    rq_activate_all_grippers(False)
    # end: URCap Program Node
    $ 3 "Wait: 10.0"
    sleep(10.0)
    # begin: URCap Program Node
    #   Source: Robotiq_Grippers, 1.8.0.1, Robotiq Inc.
    #   Type: Gripper
    $ 4 "Gripper Open (1)"
    if not(gripper_connected[0]):
      popup("Gripper 1 must be connected to run this program.", "No connection", False, True, True)
    end
    if not(rq_is_gripper_activated("1")):
      popup("Gripper 1 is not activated. Go to Installation tab > Gripper to activate it and run the program again.", "Not activated", False, True, True)
    end
    rq_set_pos_spd_for(0, 41, 66, "1")
    rq_wait_pos_spe_for_request(0, 41, 66, "1")
    rq_go_to("1")
    rq_wait("1")
    # end: URCap Program Node
    $ 5 "Loop 20 times"
    Loop_1 = 0
    while (Loop_1 < 20):
      $ 6 "MoveJ"
      $ 7 "start_position"
      movej(get_inverse_kin(p[.170260721946, .070237990876, .680621912575, .161854371436, 1.656832500967, -.237542251413], qnear=[-3.4132304827319544, -1.5469310919391077, 0.21133089065551758, -1.7181108633624476, -1.552213493977682, 7.7919034401523035]), a=1.3962634015954636, v=1.0471975511965976)
      $ 8 "MoveJ"
      $ 9 "backcase_pos"
      movej(get_inverse_kin(p[.279895687381, -.152872741101, .176453276827, .147115205195, -3.063448562531, .021495505714], qnear=[-3.980655018483297, -1.3704388777362269, 2.021009922027588, -2.1860244909869593, -1.6399787108050745, 6.916248623524801]), a=1.3962634015954636, v=1.0471975511965976)
      # begin: URCap Program Node
      #   Source: Robotiq_Grippers, 1.8.0.1, Robotiq Inc.
      #   Type: Gripper
      $ 10 "Gripper Close (1)"
      if not(gripper_connected[0]):
        popup("Gripper 1 must be connected to run this program.", "No connection", False, True, True)
      end
      if not(rq_is_gripper_activated("1")):
        popup("Gripper 1 is not activated. Go to Installation tab > Gripper to activate it and run the program again.", "Not activated", False, True, True)
      end
      rq_set_pos_spd_for(255, 41, 66, "1")
      rq_wait_pos_spe_for_request(255, 41, 66, "1")
      rq_go_to("1")
      rq_wait("1")
      # end: URCap Program Node
      # begin: URCap Program Node
      #   Source: Robotiq_Grippers, 1.8.0.1, Robotiq Inc.
      #   Type: Grip Check
      $ 11 "Grip Check"
      # begin: URCap Program Node
      #   Source: Robotiq_Grippers, 1.8.0.1, Robotiq Inc.
      #   Type: If
      $ 12 "If object detected          "
      if (rq_is_object_detected(1)):
        $ 13 "release_pos"
        movej(get_inverse_kin(p[.470773091472, .179206339821, .406393760794, -.295071821076, 2.303841954291, .069768841993], qnear=[-3.0107629934894007, -0.39652759233583623, -0.4139049688922327, -1.5799277464496058, -1.5207040945636194, 7.751115862523214]), a=1.3962634015954636, v=1.0471975511965976)
        # begin: URCap Program Node
        #   Source: Robotiq_Grippers, 1.8.0.1, Robotiq Inc.
        #   Type: Gripper
        $ 14 "Gripper Open (1)"
        if not(gripper_connected[0]):
          popup("Gripper 1 must be connected to run this program.", "No connection", False, True, True)
        end
        if not(rq_is_gripper_activated("1")):
          popup("Gripper 1 is not activated. Go to Installation tab > Gripper to activate it and run the program again.", "Not activated", False, True, True)
        end
        rq_set_pos_spd_for(0, 66, 41, "1")
        rq_wait_pos_spe_for_request(0, 66, 41, "1")
        rq_go_to("1")
        rq_wait("1")
        # end: URCap Program Node
        # end: URCap Program Node
        # begin: URCap Program Node
        #   Source: Robotiq_Grippers, 1.8.0.1, Robotiq Inc.
        #   Type: Else
        $ 15 "Else"
      else:
        # begin: URCap Program Node
        #   Source: Robotiq_Grippers, 1.8.0.1, Robotiq Inc.
        #   Type: Gripper
        $ 16 "Gripper Open (1)"
        if not(gripper_connected[0]):
          popup("Gripper 1 must be connected to run this program.", "No connection", False, True, True)
        end
        if not(rq_is_gripper_activated("1")):
          popup("Gripper 1 is not activated. Go to Installation tab > Gripper to activate it and run the program again.", "Not activated", False, True, True)
        end
        rq_set_pos_spd_for(0, 66, 41, "1")
        rq_wait_pos_spe_for_request(0, 66, 41, "1")
        rq_go_to("1")
        rq_wait("1")
        # end: URCap Program Node
        # begin: URCap Program Node
        #   Source: Robotiq_Grippers, 1.8.0.1, Robotiq Inc.
        #   Type: Gripper
        $ 17 "Gripper Close (1)"
        if not(gripper_connected[0]):
          popup("Gripper 1 must be connected to run this program.", "No connection", False, True, True)
        end
        if not(rq_is_gripper_activated("1")):
          popup("Gripper 1 is not activated. Go to Installation tab > Gripper to activate it and run the program again.", "Not activated", False, True, True)
        end
        rq_set_pos_spd_for(255, 66, 41, "1")
        rq_wait_pos_spe_for_request(255, 66, 41, "1")
        rq_go_to("1")
        rq_wait("1")
        # end: URCap Program Node
        # begin: URCap Program Node
        #   Source: Robotiq_Grippers, 1.8.0.1, Robotiq Inc.
        #   Type: Grip Check
        $ 18 "Grip Check"
        # begin: URCap Program Node
        #   Source: Robotiq_Grippers, 1.8.0.1, Robotiq Inc.
        #   Type: If
        $ 19 "If object detected          "
        if (rq_is_object_detected(1)):
          $ 20 "release_pos"
          movej(get_inverse_kin(p[.470773091472, .179206339821, .406393760794, -.295071821076, 2.303841954291, .069768841993], qnear=[-3.0107629934894007, -0.39652759233583623, -0.4139049688922327, -1.5799277464496058, -1.5207040945636194, 7.751115862523214]), a=1.3962634015954636, v=1.0471975511965976)
          # begin: URCap Program Node
          #   Source: Robotiq_Grippers, 1.8.0.1, Robotiq Inc.
          #   Type: Gripper
          $ 21 "Gripper Open (1)"
          if not(gripper_connected[0]):
            popup("Gripper 1 must be connected to run this program.", "No connection", False, True, True)
          end
          if not(rq_is_gripper_activated("1")):
            popup("Gripper 1 is not activated. Go to Installation tab > Gripper to activate it and run the program again.", "Not activated", False, True, True)
          end
          rq_set_pos_spd_for(0, 66, 41, "1")
          rq_wait_pos_spe_for_request(0, 66, 41, "1")
          rq_go_to("1")
          rq_wait("1")
          # end: URCap Program Node
          # end: URCap Program Node
          # begin: URCap Program Node
          #   Source: Robotiq_Grippers, 1.8.0.1, Robotiq Inc.
          #   Type: Else
          $ 22 "Else"
        else:
          # begin: URCap Program Node
          #   Source: Robotiq_Grippers, 1.8.0.1, Robotiq Inc.
          #   Type: Gripper
          $ 23 "Gripper Open (1)"
          if not(gripper_connected[0]):
            popup("Gripper 1 must be connected to run this program.", "No connection", False, True, True)
          end
          if not(rq_is_gripper_activated("1")):
            popup("Gripper 1 is not activated. Go to Installation tab > Gripper to activate it and run the program again.", "Not activated", False, True, True)
          end
          rq_set_pos_spd_for(0, 66, 41, "1")
          rq_wait_pos_spe_for_request(0, 66, 41, "1")
          rq_go_to("1")
          rq_wait("1")
          # end: URCap Program Node
          $ 24 "Popup"
          popup("Backcase not detected, please place in first slot", "Error", False, True, blocking=True)
          # begin: URCap Program Node
          #   Source: Robotiq_Grippers, 1.8.0.1, Robotiq Inc.
          #   Type: Gripper
          $ 25 "Gripper Close (1)"
          if not(gripper_connected[0]):
            popup("Gripper 1 must be connected to run this program.", "No connection", False, True, True)
          end
          if not(rq_is_gripper_activated("1")):
            popup("Gripper 1 is not activated. Go to Installation tab > Gripper to activate it and run the program again.", "Not activated", False, True, True)
          end
          rq_set_pos_spd_for(255, 66, 41, "1")
          rq_wait_pos_spe_for_request(255, 66, 41, "1")
          rq_go_to("1")
          rq_wait("1")
          # end: URCap Program Node
          # begin: URCap Program Node
          #   Source: Robotiq_Grippers, 1.8.0.1, Robotiq Inc.
          #   Type: Grip Check
          $ 26 "Grip Check"
          # begin: URCap Program Node
          #   Source: Robotiq_Grippers, 1.8.0.1, Robotiq Inc.
          #   Type: If
          $ 27 "If object detected          "
          if (rq_is_object_detected(1)):
            $ 28 "release_pos"
            movej(get_inverse_kin(p[.470773091472, .179206339821, .406393760794, -.295071821076, 2.303841954291, .069768841993], qnear=[-3.0107629934894007, -0.39652759233583623, -0.4139049688922327, -1.5799277464496058, -1.5207040945636194, 7.751115862523214]), a=1.3962634015954636, v=1.0471975511965976)
            # begin: URCap Program Node
            #   Source: Robotiq_Grippers, 1.8.0.1, Robotiq Inc.
            #   Type: Gripper
            $ 29 "Gripper Open (1)"
            if not(gripper_connected[0]):
              popup("Gripper 1 must be connected to run this program.", "No connection", False, True, True)
            end
            if not(rq_is_gripper_activated("1")):
              popup("Gripper 1 is not activated. Go to Installation tab > Gripper to activate it and run the program again.", "Not activated", False, True, True)
            end
            rq_set_pos_spd_for(0, 66, 41, "1")
            rq_wait_pos_spe_for_request(0, 66, 41, "1")
            rq_go_to("1")
            rq_wait("1")
            # end: URCap Program Node
            # end: URCap Program Node
            # begin: URCap Program Node
            #   Source: Robotiq_Grippers, 1.8.0.1, Robotiq Inc.
            #   Type: Else
            $ 30 "Else"
          else:
            # begin: URCap Program Node
            #   Source: Robotiq_Grippers, 1.8.0.1, Robotiq Inc.
            #   Type: Gripper
            $ 31 "Gripper Open (1)"
            if not(gripper_connected[0]):
              popup("Gripper 1 must be connected to run this program.", "No connection", False, True, True)
            end
            if not(rq_is_gripper_activated("1")):
              popup("Gripper 1 is not activated. Go to Installation tab > Gripper to activate it and run the program again.", "Not activated", False, True, True)
            end
            rq_set_pos_spd_for(0, 66, 41, "1")
            rq_wait_pos_spe_for_request(0, 66, 41, "1")
            rq_go_to("1")
            rq_wait("1")
            # end: URCap Program Node
            # begin: URCap Program Node
            #   Source: Robotiq_Grippers, 1.8.0.1, Robotiq Inc.
            #   Type: Gripper
            $ 32 "Gripper Close (1)"
            if not(gripper_connected[0]):
              popup("Gripper 1 must be connected to run this program.", "No connection", False, True, True)
            end
            if not(rq_is_gripper_activated("1")):
              popup("Gripper 1 is not activated. Go to Installation tab > Gripper to activate it and run the program again.", "Not activated", False, True, True)
            end
            rq_set_pos_spd_for(255, 66, 41, "1")
            rq_wait_pos_spe_for_request(255, 66, 41, "1")
            rq_go_to("1")
            rq_wait("1")
            # end: URCap Program Node
            # begin: URCap Program Node
            #   Source: Robotiq_Grippers, 1.8.0.1, Robotiq Inc.
            #   Type: Grip Check
            $ 33 "Grip Check"
            # begin: URCap Program Node
            #   Source: Robotiq_Grippers, 1.8.0.1, Robotiq Inc.
            #   Type: If
            $ 34 "If object detected          "
            if (rq_is_object_detected(1)):
              $ 35 "release_pos"
              movej(get_inverse_kin(p[.470773091472, .179206339821, .406393760794, -.295071821076, 2.303841954291, .069768841993], qnear=[-3.0107629934894007, -0.39652759233583623, -0.4139049688922327, -1.5799277464496058, -1.5207040945636194, 7.751115862523214]), a=1.3962634015954636, v=1.0471975511965976)
              # begin: URCap Program Node
              #   Source: Robotiq_Grippers, 1.8.0.1, Robotiq Inc.
              #   Type: Gripper
              $ 36 "Gripper Open (1)"
              if not(gripper_connected[0]):
                popup("Gripper 1 must be connected to run this program.", "No connection", False, True, True)
              end
              if not(rq_is_gripper_activated("1")):
                popup("Gripper 1 is not activated. Go to Installation tab > Gripper to activate it and run the program again.", "Not activated", False, True, True)
              end
              rq_set_pos_spd_for(0, 66, 41, "1")
              rq_wait_pos_spe_for_request(0, 66, 41, "1")
              rq_go_to("1")
              rq_wait("1")
              # end: URCap Program Node
              # end: URCap Program Node
              # begin: URCap Program Node
              #   Source: Robotiq_Grippers, 1.8.0.1, Robotiq Inc.
              #   Type: Else
              $ 37 "Else"
            else:
              # begin: URCap Program Node
              #   Source: Robotiq_Grippers, 1.8.0.1, Robotiq Inc.
              #   Type: Gripper
              $ 38 "Gripper Open (1)"
              if not(gripper_connected[0]):
                popup("Gripper 1 must be connected to run this program.", "No connection", False, True, True)
              end
              if not(rq_is_gripper_activated("1")):
                popup("Gripper 1 is not activated. Go to Installation tab > Gripper to activate it and run the program again.", "Not activated", False, True, True)
              end
              rq_set_pos_spd_for(0, 66, 41, "1")
              rq_wait_pos_spe_for_request(0, 66, 41, "1")
              rq_go_to("1")
              rq_wait("1")
              # end: URCap Program Node
              $ 39 "Halt"
              halt
              # end: URCap Program Node
            end
            # end: URCap Program Node
            # end: URCap Program Node
          end
          # end: URCap Program Node
          # end: URCap Program Node
        end
        # end: URCap Program Node
        # end: URCap Program Node
      end
      # end: URCap Program Node
      $ 40 "MoveJ"
      $ 41 "pcb_pos"
      movej(get_inverse_kin(p[.267160343869, -.023216767798, .195523930932, .156439806997, -3.068996142090, .012381886328], qnear=[-3.6437318960772913, -1.6386993567096155, 2.196641445159912, -2.0753896872149866, -1.6169927755938929, 7.247925941144125]), a=1.3962634015954636, v=1.0471975511965976)
      # begin: URCap Program Node
      #   Source: Robotiq_Grippers, 1.8.0.1, Robotiq Inc.
      #   Type: Gripper
      $ 42 "Gripper Close (1)"
      if not(gripper_connected[0]):
        popup("Gripper 1 must be connected to run this program.", "No connection", False, True, True)
      end
      if not(rq_is_gripper_activated("1")):
        popup("Gripper 1 is not activated. Go to Installation tab > Gripper to activate it and run the program again.", "Not activated", False, True, True)
      end
      rq_set_pos_spd_for(255, 41, 66, "1")
      rq_wait_pos_spe_for_request(255, 41, 66, "1")
      rq_go_to("1")
      rq_wait("1")
      # end: URCap Program Node
      # begin: URCap Program Node
      #   Source: Robotiq_Grippers, 1.8.0.1, Robotiq Inc.
      #   Type: Grip Check
      $ 43 "Grip Check"
      # begin: URCap Program Node
      #   Source: Robotiq_Grippers, 1.8.0.1, Robotiq Inc.
      #   Type: If
      $ 44 "If object detected          "
      if (rq_is_object_detected(1)):
        $ 45 "release_pos"
        movej(get_inverse_kin(p[.470773091472, .179206339821, .406393760794, -.295071821076, 2.303841954291, .069768841993], qnear=[-3.0107629934894007, -0.39652759233583623, -0.4139049688922327, -1.5799277464496058, -1.5207040945636194, 7.751115862523214]), a=1.3962634015954636, v=1.0471975511965976)
        # begin: URCap Program Node
        #   Source: Robotiq_Grippers, 1.8.0.1, Robotiq Inc.
        #   Type: Gripper
        $ 46 "Gripper Open (1)"
        if not(gripper_connected[0]):
          popup("Gripper 1 must be connected to run this program.", "No connection", False, True, True)
        end
        if not(rq_is_gripper_activated("1")):
          popup("Gripper 1 is not activated. Go to Installation tab > Gripper to activate it and run the program again.", "Not activated", False, True, True)
        end
        rq_set_pos_spd_for(0, 66, 41, "1")
        rq_wait_pos_spe_for_request(0, 66, 41, "1")
        rq_go_to("1")
        rq_wait("1")
        # end: URCap Program Node
        # end: URCap Program Node
        # begin: URCap Program Node
        #   Source: Robotiq_Grippers, 1.8.0.1, Robotiq Inc.
        #   Type: Else
        $ 47 "Else"
      else:
        # begin: URCap Program Node
        #   Source: Robotiq_Grippers, 1.8.0.1, Robotiq Inc.
        #   Type: Gripper
        $ 48 "Gripper Open (1)"
        if not(gripper_connected[0]):
          popup("Gripper 1 must be connected to run this program.", "No connection", False, True, True)
        end
        if not(rq_is_gripper_activated("1")):
          popup("Gripper 1 is not activated. Go to Installation tab > Gripper to activate it and run the program again.", "Not activated", False, True, True)
        end
        rq_set_pos_spd_for(0, 66, 41, "1")
        rq_wait_pos_spe_for_request(0, 66, 41, "1")
        rq_go_to("1")
        rq_wait("1")
        # end: URCap Program Node
        $ 49 "Popup"
        popup("PCB not detected, please place in second slot", "Error", False, True, blocking=True)
        # begin: URCap Program Node
        #   Source: Robotiq_Grippers, 1.8.0.1, Robotiq Inc.
        #   Type: Gripper
        $ 50 "Gripper Close (1)"
        if not(gripper_connected[0]):
          popup("Gripper 1 must be connected to run this program.", "No connection", False, True, True)
        end
        if not(rq_is_gripper_activated("1")):
          popup("Gripper 1 is not activated. Go to Installation tab > Gripper to activate it and run the program again.", "Not activated", False, True, True)
        end
        rq_set_pos_spd_for(255, 66, 41, "1")
        rq_wait_pos_spe_for_request(255, 66, 41, "1")
        rq_go_to("1")
        rq_wait("1")
        # end: URCap Program Node
        # begin: URCap Program Node
        #   Source: Robotiq_Grippers, 1.8.0.1, Robotiq Inc.
        #   Type: Grip Check
        $ 51 "Grip Check"
        # begin: URCap Program Node
        #   Source: Robotiq_Grippers, 1.8.0.1, Robotiq Inc.
        #   Type: If
        $ 52 "If object detected          "
        if (rq_is_object_detected(1)):
          $ 53 "release_pos"
          movej(get_inverse_kin(p[.470773091472, .179206339821, .406393760794, -.295071821076, 2.303841954291, .069768841993], qnear=[-3.0107629934894007, -0.39652759233583623, -0.4139049688922327, -1.5799277464496058, -1.5207040945636194, 7.751115862523214]), a=1.3962634015954636, v=1.0471975511965976)
          # begin: URCap Program Node
          #   Source: Robotiq_Grippers, 1.8.0.1, Robotiq Inc.
          #   Type: Gripper
          $ 54 "Gripper Open (1)"
          if not(gripper_connected[0]):
            popup("Gripper 1 must be connected to run this program.", "No connection", False, True, True)
          end
          if not(rq_is_gripper_activated("1")):
            popup("Gripper 1 is not activated. Go to Installation tab > Gripper to activate it and run the program again.", "Not activated", False, True, True)
          end
          rq_set_pos_spd_for(0, 66, 41, "1")
          rq_wait_pos_spe_for_request(0, 66, 41, "1")
          rq_go_to("1")
          rq_wait("1")
          # end: URCap Program Node
          # end: URCap Program Node
          # begin: URCap Program Node
          #   Source: Robotiq_Grippers, 1.8.0.1, Robotiq Inc.
          #   Type: Else
          $ 55 "Else"
        else:
          # begin: URCap Program Node
          #   Source: Robotiq_Grippers, 1.8.0.1, Robotiq Inc.
          #   Type: Gripper
          $ 56 "Gripper Open (1)"
          if not(gripper_connected[0]):
            popup("Gripper 1 must be connected to run this program.", "No connection", False, True, True)
          end
          if not(rq_is_gripper_activated("1")):
            popup("Gripper 1 is not activated. Go to Installation tab > Gripper to activate it and run the program again.", "Not activated", False, True, True)
          end
          rq_set_pos_spd_for(0, 66, 41, "1")
          rq_wait_pos_spe_for_request(0, 66, 41, "1")
          rq_go_to("1")
          rq_wait("1")
          # end: URCap Program Node
          # begin: URCap Program Node
          #   Source: Robotiq_Grippers, 1.8.0.1, Robotiq Inc.
          #   Type: Gripper
          $ 57 "Gripper Close (1)"
          if not(gripper_connected[0]):
            popup("Gripper 1 must be connected to run this program.", "No connection", False, True, True)
          end
          if not(rq_is_gripper_activated("1")):
            popup("Gripper 1 is not activated. Go to Installation tab > Gripper to activate it and run the program again.", "Not activated", False, True, True)
          end
          rq_set_pos_spd_for(255, 66, 41, "1")
          rq_wait_pos_spe_for_request(255, 66, 41, "1")
          rq_go_to("1")
          rq_wait("1")
          # end: URCap Program Node
          # begin: URCap Program Node
          #   Source: Robotiq_Grippers, 1.8.0.1, Robotiq Inc.
          #   Type: Grip Check
          $ 58 "Grip Check"
          # begin: URCap Program Node
          #   Source: Robotiq_Grippers, 1.8.0.1, Robotiq Inc.
          #   Type: If
          $ 59 "If object detected          "
          if (rq_is_object_detected(1)):
            $ 60 "release_pos"
            movej(get_inverse_kin(p[.470773091472, .179206339821, .406393760794, -.295071821076, 2.303841954291, .069768841993], qnear=[-3.0107629934894007, -0.39652759233583623, -0.4139049688922327, -1.5799277464496058, -1.5207040945636194, 7.751115862523214]), a=1.3962634015954636, v=1.0471975511965976)
            # begin: URCap Program Node
            #   Source: Robotiq_Grippers, 1.8.0.1, Robotiq Inc.
            #   Type: Gripper
            $ 61 "Gripper Open (1)"
            if not(gripper_connected[0]):
              popup("Gripper 1 must be connected to run this program.", "No connection", False, True, True)
            end
            if not(rq_is_gripper_activated("1")):
              popup("Gripper 1 is not activated. Go to Installation tab > Gripper to activate it and run the program again.", "Not activated", False, True, True)
            end
            rq_set_pos_spd_for(0, 66, 41, "1")
            rq_wait_pos_spe_for_request(0, 66, 41, "1")
            rq_go_to("1")
            rq_wait("1")
            # end: URCap Program Node
            # end: URCap Program Node
            # begin: URCap Program Node
            #   Source: Robotiq_Grippers, 1.8.0.1, Robotiq Inc.
            #   Type: Else
            $ 62 "Else"
          else:
            # begin: URCap Program Node
            #   Source: Robotiq_Grippers, 1.8.0.1, Robotiq Inc.
            #   Type: Gripper
            $ 63 "Gripper Open (1)"
            if not(gripper_connected[0]):
              popup("Gripper 1 must be connected to run this program.", "No connection", False, True, True)
            end
            if not(rq_is_gripper_activated("1")):
              popup("Gripper 1 is not activated. Go to Installation tab > Gripper to activate it and run the program again.", "Not activated", False, True, True)
            end
            rq_set_pos_spd_for(0, 66, 41, "1")
            rq_wait_pos_spe_for_request(0, 66, 41, "1")
            rq_go_to("1")
            rq_wait("1")
            # end: URCap Program Node
            # begin: URCap Program Node
            #   Source: Robotiq_Grippers, 1.8.0.1, Robotiq Inc.
            #   Type: Gripper
            $ 64 "Gripper Close (1)"
            if not(gripper_connected[0]):
              popup("Gripper 1 must be connected to run this program.", "No connection", False, True, True)
            end
            if not(rq_is_gripper_activated("1")):
              popup("Gripper 1 is not activated. Go to Installation tab > Gripper to activate it and run the program again.", "Not activated", False, True, True)
            end
            rq_set_pos_spd_for(255, 66, 41, "1")
            rq_wait_pos_spe_for_request(255, 66, 41, "1")
            rq_go_to("1")
            rq_wait("1")
            # end: URCap Program Node
            # begin: URCap Program Node
            #   Source: Robotiq_Grippers, 1.8.0.1, Robotiq Inc.
            #   Type: Grip Check
            $ 65 "Grip Check"
            # begin: URCap Program Node
            #   Source: Robotiq_Grippers, 1.8.0.1, Robotiq Inc.
            #   Type: If
            $ 66 "If object detected          "
            if (rq_is_object_detected(1)):
              $ 67 "release_pos"
              movej(get_inverse_kin(p[.470773091472, .179206339821, .406393760794, -.295071821076, 2.303841954291, .069768841993], qnear=[-3.0107629934894007, -0.39652759233583623, -0.4139049688922327, -1.5799277464496058, -1.5207040945636194, 7.751115862523214]), a=1.3962634015954636, v=1.0471975511965976)
              # begin: URCap Program Node
              #   Source: Robotiq_Grippers, 1.8.0.1, Robotiq Inc.
              #   Type: Gripper
              $ 68 "Gripper Open (1)"
              if not(gripper_connected[0]):
                popup("Gripper 1 must be connected to run this program.", "No connection", False, True, True)
              end
              if not(rq_is_gripper_activated("1")):
                popup("Gripper 1 is not activated. Go to Installation tab > Gripper to activate it and run the program again.", "Not activated", False, True, True)
              end
              rq_set_pos_spd_for(0, 66, 41, "1")
              rq_wait_pos_spe_for_request(0, 66, 41, "1")
              rq_go_to("1")
              rq_wait("1")
              # end: URCap Program Node
              # end: URCap Program Node
              # begin: URCap Program Node
              #   Source: Robotiq_Grippers, 1.8.0.1, Robotiq Inc.
              #   Type: Else
              $ 69 "Else"
            else:
              # begin: URCap Program Node
              #   Source: Robotiq_Grippers, 1.8.0.1, Robotiq Inc.
              #   Type: Gripper
              $ 70 "Gripper Open (1)"
              if not(gripper_connected[0]):
                popup("Gripper 1 must be connected to run this program.", "No connection", False, True, True)
              end
              if not(rq_is_gripper_activated("1")):
                popup("Gripper 1 is not activated. Go to Installation tab > Gripper to activate it and run the program again.", "Not activated", False, True, True)
              end
              rq_set_pos_spd_for(0, 66, 41, "1")
              rq_wait_pos_spe_for_request(0, 66, 41, "1")
              rq_go_to("1")
              rq_wait("1")
              # end: URCap Program Node
              $ 71 "Halt"
              halt
              # end: URCap Program Node
            end
            # end: URCap Program Node
            # end: URCap Program Node
          end
          # end: URCap Program Node
          # end: URCap Program Node
        end
        # end: URCap Program Node
        # end: URCap Program Node
      end
      # end: URCap Program Node
      $ 72 "MoveJ"
      $ 73 "frontcase_pos"
      movej(get_inverse_kin(p[.268774768307, .107599353393, .176019128009, .147391443851, -3.063198716239, .021669865685], qnear=[-3.151196066533224, -1.4895699659930628, 2.1479902267456055, -2.1561153570758265, -1.5922024885760706, 7.745294515286581]), a=1.3962634015954636, v=1.0471975511965976)
      # begin: URCap Program Node
      #   Source: Robotiq_Grippers, 1.8.0.1, Robotiq Inc.
      #   Type: Gripper
      $ 74 "Gripper Close (1)"
      if not(gripper_connected[0]):
        popup("Gripper 1 must be connected to run this program.", "No connection", False, True, True)
      end
      if not(rq_is_gripper_activated("1")):
        popup("Gripper 1 is not activated. Go to Installation tab > Gripper to activate it and run the program again.", "Not activated", False, True, True)
      end
      rq_set_pos_spd_for(255, 66, 41, "1")
      rq_wait_pos_spe_for_request(255, 66, 41, "1")
      rq_go_to("1")
      rq_wait("1")
      # end: URCap Program Node
      # begin: URCap Program Node
      #   Source: Robotiq_Grippers, 1.8.0.1, Robotiq Inc.
      #   Type: Grip Check
      $ 75 "Grip Check"
      # begin: URCap Program Node
      #   Source: Robotiq_Grippers, 1.8.0.1, Robotiq Inc.
      #   Type: If
      $ 76 "If object detected          "
      if (rq_is_object_detected(1)):
        $ 77 "release_pos"
        movej(get_inverse_kin(p[.470773091472, .179206339821, .406393760794, -.295071821076, 2.303841954291, .069768841993], qnear=[-3.0107629934894007, -0.39652759233583623, -0.4139049688922327, -1.5799277464496058, -1.5207040945636194, 7.751115862523214]), a=1.3962634015954636, v=1.0471975511965976)
        # begin: URCap Program Node
        #   Source: Robotiq_Grippers, 1.8.0.1, Robotiq Inc.
        #   Type: Gripper
        $ 78 "Gripper Open (1)"
        if not(gripper_connected[0]):
          popup("Gripper 1 must be connected to run this program.", "No connection", False, True, True)
        end
        if not(rq_is_gripper_activated("1")):
          popup("Gripper 1 is not activated. Go to Installation tab > Gripper to activate it and run the program again.", "Not activated", False, True, True)
        end
        rq_set_pos_spd_for(0, 66, 41, "1")
        rq_wait_pos_spe_for_request(0, 66, 41, "1")
        rq_go_to("1")
        rq_wait("1")
        # end: URCap Program Node
        # end: URCap Program Node
        # begin: URCap Program Node
        #   Source: Robotiq_Grippers, 1.8.0.1, Robotiq Inc.
        #   Type: Else
        $ 79 "Else"
      else:
        # begin: URCap Program Node
        #   Source: Robotiq_Grippers, 1.8.0.1, Robotiq Inc.
        #   Type: Gripper
        $ 80 "Gripper Open (1)"
        if not(gripper_connected[0]):
          popup("Gripper 1 must be connected to run this program.", "No connection", False, True, True)
        end
        if not(rq_is_gripper_activated("1")):
          popup("Gripper 1 is not activated. Go to Installation tab > Gripper to activate it and run the program again.", "Not activated", False, True, True)
        end
        rq_set_pos_spd_for(0, 66, 41, "1")
        rq_wait_pos_spe_for_request(0, 66, 41, "1")
        rq_go_to("1")
        rq_wait("1")
        # end: URCap Program Node
        $ 81 "Popup"
        popup("Frontcase not detected, please place in third slot", "Error", False, True, blocking=True)
        # begin: URCap Program Node
        #   Source: Robotiq_Grippers, 1.8.0.1, Robotiq Inc.
        #   Type: Gripper
        $ 82 "Gripper Close (1)"
        if not(gripper_connected[0]):
          popup("Gripper 1 must be connected to run this program.", "No connection", False, True, True)
        end
        if not(rq_is_gripper_activated("1")):
          popup("Gripper 1 is not activated. Go to Installation tab > Gripper to activate it and run the program again.", "Not activated", False, True, True)
        end
        rq_set_pos_spd_for(255, 66, 41, "1")
        rq_wait_pos_spe_for_request(255, 66, 41, "1")
        rq_go_to("1")
        rq_wait("1")
        # end: URCap Program Node
        # begin: URCap Program Node
        #   Source: Robotiq_Grippers, 1.8.0.1, Robotiq Inc.
        #   Type: Grip Check
        $ 83 "Grip Check"
        # begin: URCap Program Node
        #   Source: Robotiq_Grippers, 1.8.0.1, Robotiq Inc.
        #   Type: If
        $ 84 "If object detected          "
        if (rq_is_object_detected(1)):
          $ 85 "release_pos"
          movej(get_inverse_kin(p[.470773091472, .179206339821, .406393760794, -.295071821076, 2.303841954291, .069768841993], qnear=[-3.0107629934894007, -0.39652759233583623, -0.4139049688922327, -1.5799277464496058, -1.5207040945636194, 7.751115862523214]), a=1.3962634015954636, v=1.0471975511965976)
          # begin: URCap Program Node
          #   Source: Robotiq_Grippers, 1.8.0.1, Robotiq Inc.
          #   Type: Gripper
          $ 86 "Gripper Open (1)"
          if not(gripper_connected[0]):
            popup("Gripper 1 must be connected to run this program.", "No connection", False, True, True)
          end
          if not(rq_is_gripper_activated("1")):
            popup("Gripper 1 is not activated. Go to Installation tab > Gripper to activate it and run the program again.", "Not activated", False, True, True)
          end
          rq_set_pos_spd_for(0, 66, 41, "1")
          rq_wait_pos_spe_for_request(0, 66, 41, "1")
          rq_go_to("1")
          rq_wait("1")
          # end: URCap Program Node
          # end: URCap Program Node
          # begin: URCap Program Node
          #   Source: Robotiq_Grippers, 1.8.0.1, Robotiq Inc.
          #   Type: Else
          $ 87 "Else"
        else:
          # begin: URCap Program Node
          #   Source: Robotiq_Grippers, 1.8.0.1, Robotiq Inc.
          #   Type: Gripper
          $ 88 "Gripper Open (1)"
          if not(gripper_connected[0]):
            popup("Gripper 1 must be connected to run this program.", "No connection", False, True, True)
          end
          if not(rq_is_gripper_activated("1")):
            popup("Gripper 1 is not activated. Go to Installation tab > Gripper to activate it and run the program again.", "Not activated", False, True, True)
          end
          rq_set_pos_spd_for(0, 66, 41, "1")
          rq_wait_pos_spe_for_request(0, 66, 41, "1")
          rq_go_to("1")
          rq_wait("1")
          # end: URCap Program Node
          # begin: URCap Program Node
          #   Source: Robotiq_Grippers, 1.8.0.1, Robotiq Inc.
          #   Type: Gripper
          $ 89 "Gripper Close (1)"
          if not(gripper_connected[0]):
            popup("Gripper 1 must be connected to run this program.", "No connection", False, True, True)
          end
          if not(rq_is_gripper_activated("1")):
            popup("Gripper 1 is not activated. Go to Installation tab > Gripper to activate it and run the program again.", "Not activated", False, True, True)
          end
          rq_set_pos_spd_for(255, 66, 41, "1")
          rq_wait_pos_spe_for_request(255, 66, 41, "1")
          rq_go_to("1")
          rq_wait("1")
          # end: URCap Program Node
          # begin: URCap Program Node
          #   Source: Robotiq_Grippers, 1.8.0.1, Robotiq Inc.
          #   Type: Grip Check
          $ 90 "Grip Check"
          # begin: URCap Program Node
          #   Source: Robotiq_Grippers, 1.8.0.1, Robotiq Inc.
          #   Type: If
          $ 91 "If object detected          "
          if (rq_is_object_detected(1)):
            $ 92 "release_pos"
            movej(get_inverse_kin(p[.470773091472, .179206339821, .406393760794, -.295071821076, 2.303841954291, .069768841993], qnear=[-3.0107629934894007, -0.39652759233583623, -0.4139049688922327, -1.5799277464496058, -1.5207040945636194, 7.751115862523214]), a=1.3962634015954636, v=1.0471975511965976)
            # begin: URCap Program Node
            #   Source: Robotiq_Grippers, 1.8.0.1, Robotiq Inc.
            #   Type: Gripper
            $ 93 "Gripper Open (1)"
            if not(gripper_connected[0]):
              popup("Gripper 1 must be connected to run this program.", "No connection", False, True, True)
            end
            if not(rq_is_gripper_activated("1")):
              popup("Gripper 1 is not activated. Go to Installation tab > Gripper to activate it and run the program again.", "Not activated", False, True, True)
            end
            rq_set_pos_spd_for(0, 66, 41, "1")
            rq_wait_pos_spe_for_request(0, 66, 41, "1")
            rq_go_to("1")
            rq_wait("1")
            # end: URCap Program Node
            # end: URCap Program Node
            # begin: URCap Program Node
            #   Source: Robotiq_Grippers, 1.8.0.1, Robotiq Inc.
            #   Type: Else
            $ 94 "Else"
          else:
            # begin: URCap Program Node
            #   Source: Robotiq_Grippers, 1.8.0.1, Robotiq Inc.
            #   Type: Gripper
            $ 95 "Gripper Open (1)"
            if not(gripper_connected[0]):
              popup("Gripper 1 must be connected to run this program.", "No connection", False, True, True)
            end
            if not(rq_is_gripper_activated("1")):
              popup("Gripper 1 is not activated. Go to Installation tab > Gripper to activate it and run the program again.", "Not activated", False, True, True)
            end
            rq_set_pos_spd_for(0, 66, 41, "1")
            rq_wait_pos_spe_for_request(0, 66, 41, "1")
            rq_go_to("1")
            rq_wait("1")
            # end: URCap Program Node
            # begin: URCap Program Node
            #   Source: Robotiq_Grippers, 1.8.0.1, Robotiq Inc.
            #   Type: Gripper
            $ 96 "Gripper Close (1)"
            if not(gripper_connected[0]):
              popup("Gripper 1 must be connected to run this program.", "No connection", False, True, True)
            end
            if not(rq_is_gripper_activated("1")):
              popup("Gripper 1 is not activated. Go to Installation tab > Gripper to activate it and run the program again.", "Not activated", False, True, True)
            end
            rq_set_pos_spd_for(255, 66, 41, "1")
            rq_wait_pos_spe_for_request(255, 66, 41, "1")
            rq_go_to("1")
            rq_wait("1")
            # end: URCap Program Node
            # begin: URCap Program Node
            #   Source: Robotiq_Grippers, 1.8.0.1, Robotiq Inc.
            #   Type: Grip Check
            $ 97 "Grip Check"
            # begin: URCap Program Node
            #   Source: Robotiq_Grippers, 1.8.0.1, Robotiq Inc.
            #   Type: If
            $ 98 "If object detected          "
            if (rq_is_object_detected(1)):
              $ 99 "release_pos"
              movej(get_inverse_kin(p[.470773091472, .179206339821, .406393760794, -.295071821076, 2.303841954291, .069768841993], qnear=[-3.0107629934894007, -0.39652759233583623, -0.4139049688922327, -1.5799277464496058, -1.5207040945636194, 7.751115862523214]), a=1.3962634015954636, v=1.0471975511965976)
              # begin: URCap Program Node
              #   Source: Robotiq_Grippers, 1.8.0.1, Robotiq Inc.
              #   Type: Gripper
              $ 100 "Gripper Open (1)"
              if not(gripper_connected[0]):
                popup("Gripper 1 must be connected to run this program.", "No connection", False, True, True)
              end
              if not(rq_is_gripper_activated("1")):
                popup("Gripper 1 is not activated. Go to Installation tab > Gripper to activate it and run the program again.", "Not activated", False, True, True)
              end
              rq_set_pos_spd_for(0, 66, 41, "1")
              rq_wait_pos_spe_for_request(0, 66, 41, "1")
              rq_go_to("1")
              rq_wait("1")
              # end: URCap Program Node
              # end: URCap Program Node
              # begin: URCap Program Node
              #   Source: Robotiq_Grippers, 1.8.0.1, Robotiq Inc.
              #   Type: Else
              $ 101 "Else"
            else:
              # begin: URCap Program Node
              #   Source: Robotiq_Grippers, 1.8.0.1, Robotiq Inc.
              #   Type: Gripper
              $ 102 "Gripper Open (1)"
              if not(gripper_connected[0]):
                popup("Gripper 1 must be connected to run this program.", "No connection", False, True, True)
              end
              if not(rq_is_gripper_activated("1")):
                popup("Gripper 1 is not activated. Go to Installation tab > Gripper to activate it and run the program again.", "Not activated", False, True, True)
              end
              rq_set_pos_spd_for(0, 66, 41, "1")
              rq_wait_pos_spe_for_request(0, 66, 41, "1")
              rq_go_to("1")
              rq_wait("1")
              # end: URCap Program Node
              $ 103 "Halt"
              halt
              # end: URCap Program Node
            end
            # end: URCap Program Node
            # end: URCap Program Node
          end
          # end: URCap Program Node
          # end: URCap Program Node
        end
        # end: URCap Program Node
        # end: URCap Program Node
      end
      # end: URCap Program Node
      $ 104 "MoveJ"
      $ 105 "start_position"
      movej(get_inverse_kin(p[.170260721946, .070237990876, .680621912575, .161854371436, 1.656832500967, -.237542251413], qnear=[-3.4132304827319544, -1.5469310919391077, 0.21133089065551758, -1.7181108633624476, -1.552213493977682, 7.7919034401523035]), a=1.3962634015954636, v=1.0471975511965976)
      $ 106 "Wait: 10.0"
      sleep(10.0)
      Loop_1 = Loop_1 + 1
    end
  end
end
